PROGRAM SP3_2_Y131
VAR
	CompareOutput131_00: CMP_OC_DW;
	CompareOutput131_01: CMP_OC_DW;
	CompareOutput131_02: CMP_OC_DW;
	CompareOutput131_03: CMP_OC_DW;
	CompareOutput131_04: CMP_OC_DW;
	CompareOutput131_05: CMP_OC_DW;
	CompareOutput131_06: CMP_OC_DW;
	CompareOutput131_07: CMP_OC_DW;
	CompareOutput131_08: CMP_OC_DW;
	CompareOutput131_09: CMP_OC_DW;
	CompareOutput131_10: CMP_OC_DW;
	CompareOutput131_11: CMP_OC_DW;
	CompareOutput131_12: CMP_OC_DW;
	CompareOutput131_13: CMP_OC_DW;
	CompareOutput131_14: CMP_OC_DW;
	CompareOutput131_15: CMP_OC_DW;

END_VAR

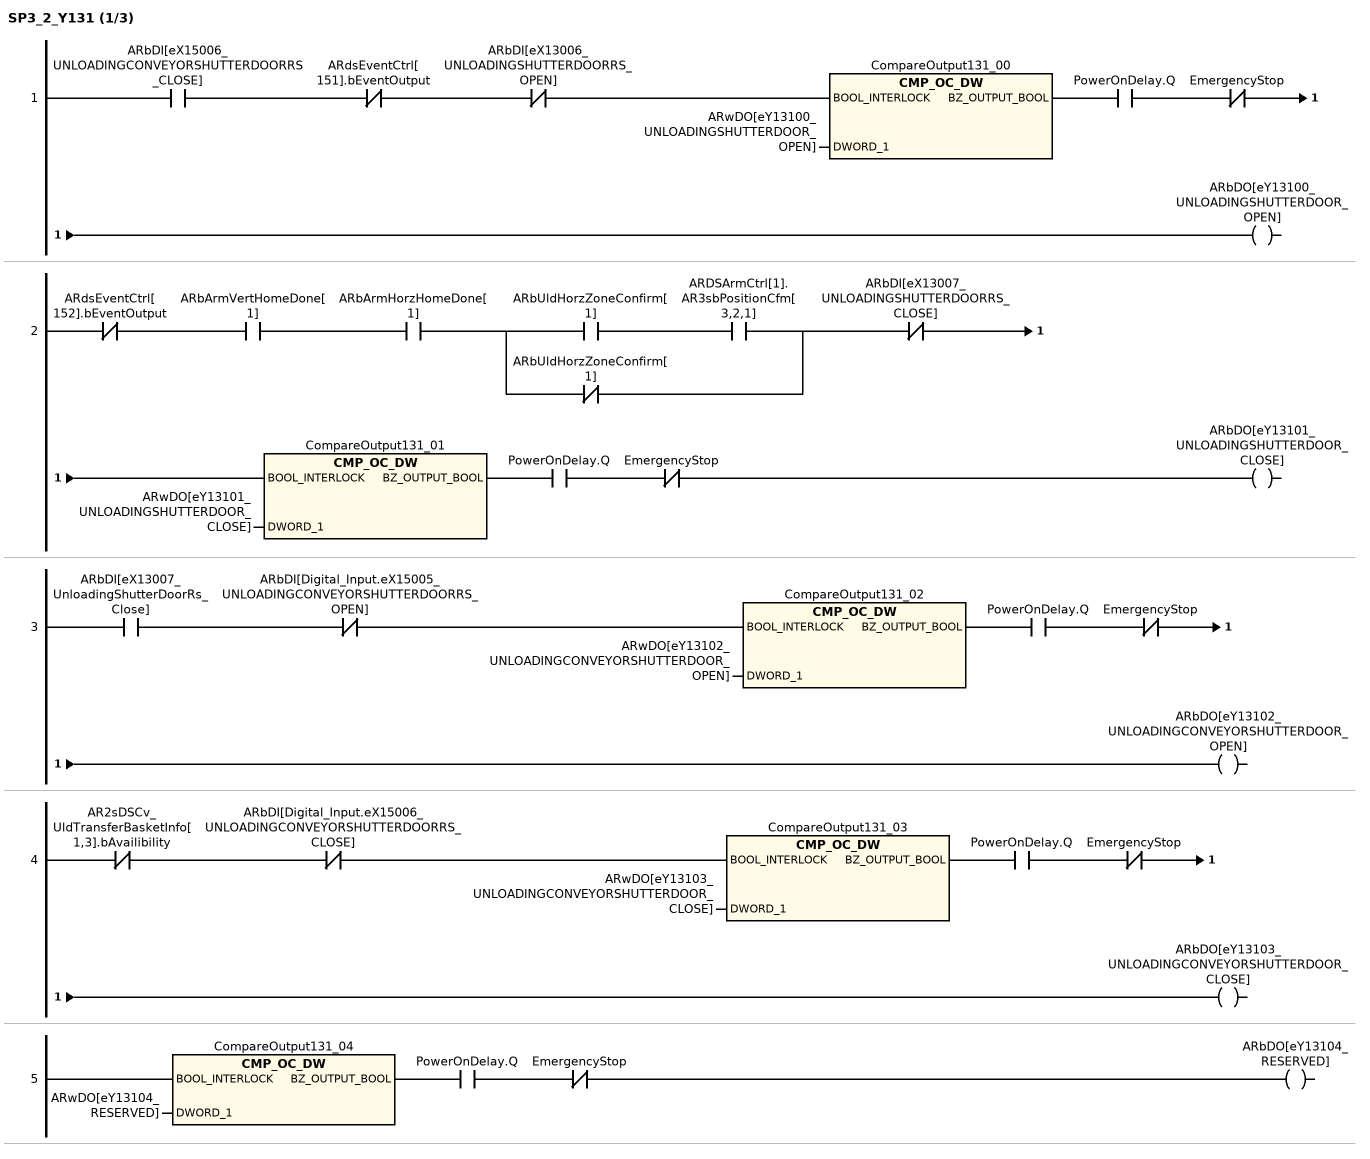
// NETWORK 1
CompareOutput131_00(BOOL_INTERLOCK := ARbDI[eX15006_UNLOADINGCONVEYORSHUTTERDOORRS_CLOSE] AND NOT ARdsEventCtrl[151].bEventOutput AND NOT ARbDI[eX13006_UNLOADINGSHUTTERDOORRS_OPEN], DWORD_1 := ARwDO[eY13100_UNLOADINGSHUTTERDOOR_OPEN]); // CMP_OC_DW
ARbDO[eY13100_UNLOADINGSHUTTERDOOR_OPEN] := CompareOutput131_00.BZ_OUTPUT_BOOL AND PowerOnDelay.Q AND NOT EmergencyStop;

// NETWORK 2
CompareOutput131_01(BOOL_INTERLOCK := NOT ARdsEventCtrl[152].bEventOutput AND ARbArmVertHomeDone[1] AND ARbArmHorzHomeDone[1] AND (ARbUldHorzZoneConfirm[1] AND ARDSArmCtrl[1].AR3sbPositionCfm[3,2,1] OR NOT ARbUldHorzZoneConfirm[1]) AND NOT ARbDI[eX13007_UNLOADINGSHUTTERDOORRS_CLOSE], DWORD_1 := ARwDO[eY13101_UNLOADINGSHUTTERDOOR_CLOSE]); // CMP_OC_DW
ARbDO[eY13101_UNLOADINGSHUTTERDOOR_CLOSE] := CompareOutput131_01.BZ_OUTPUT_BOOL AND PowerOnDelay.Q AND NOT EmergencyStop;

// NETWORK 3
CompareOutput131_02(BOOL_INTERLOCK := ARbDI[eX13007_UnloadingShutterDoorRs_Close] AND NOT ARbDI[Digital_Input.eX15005_UNLOADINGCONVEYORSHUTTERDOORRS_OPEN], DWORD_1 := ARwDO[eY13102_UNLOADINGCONVEYORSHUTTERDOOR_OPEN]); // CMP_OC_DW
ARbDO[eY13102_UNLOADINGCONVEYORSHUTTERDOOR_OPEN] := CompareOutput131_02.BZ_OUTPUT_BOOL AND PowerOnDelay.Q AND NOT EmergencyStop;

// NETWORK 4
CompareOutput131_03(BOOL_INTERLOCK := NOT AR2sDSCv_UldTransferBasketInfo[1,3].bAvailibility AND NOT ARbDI[Digital_Input.eX15006_UNLOADINGCONVEYORSHUTTERDOORRS_CLOSE], DWORD_1 := ARwDO[eY13103_UNLOADINGCONVEYORSHUTTERDOOR_CLOSE]); // CMP_OC_DW
ARbDO[eY13103_UNLOADINGCONVEYORSHUTTERDOOR_CLOSE] := CompareOutput131_03.BZ_OUTPUT_BOOL AND PowerOnDelay.Q AND NOT EmergencyStop;

// NETWORK 5
CompareOutput131_04(BOOL_INTERLOCK := TRUE, DWORD_1 := ARwDO[eY13104_RESERVED]); // CMP_OC_DW
ARbDO[eY13104_RESERVED] := CompareOutput131_04.BZ_OUTPUT_BOOL AND PowerOnDelay.Q AND NOT EmergencyStop;

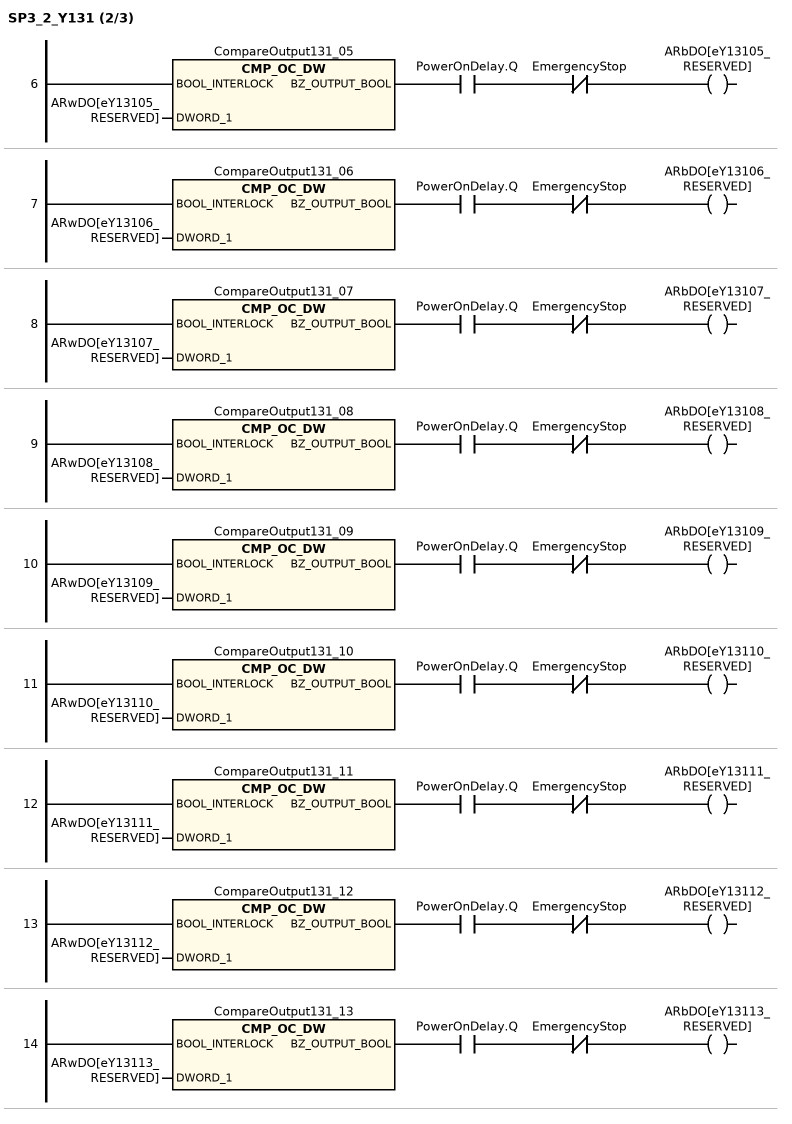
// NETWORK 6
CompareOutput131_05(BOOL_INTERLOCK := TRUE, DWORD_1 := ARwDO[eY13105_RESERVED]); // CMP_OC_DW
ARbDO[eY13105_RESERVED] := CompareOutput131_05.BZ_OUTPUT_BOOL AND PowerOnDelay.Q AND NOT EmergencyStop;

// NETWORK 7
CompareOutput131_06(BOOL_INTERLOCK := TRUE, DWORD_1 := ARwDO[eY13106_RESERVED]); // CMP_OC_DW
ARbDO[eY13106_RESERVED] := CompareOutput131_06.BZ_OUTPUT_BOOL AND PowerOnDelay.Q AND NOT EmergencyStop;

// NETWORK 8
CompareOutput131_07(BOOL_INTERLOCK := TRUE, DWORD_1 := ARwDO[eY13107_RESERVED]); // CMP_OC_DW
ARbDO[eY13107_RESERVED] := CompareOutput131_07.BZ_OUTPUT_BOOL AND PowerOnDelay.Q AND NOT EmergencyStop;

// NETWORK 9
CompareOutput131_08(BOOL_INTERLOCK := TRUE, DWORD_1 := ARwDO[eY13108_RESERVED]); // CMP_OC_DW
ARbDO[eY13108_RESERVED] := CompareOutput131_08.BZ_OUTPUT_BOOL AND PowerOnDelay.Q AND NOT EmergencyStop;

// NETWORK 10
CompareOutput131_09(BOOL_INTERLOCK := TRUE, DWORD_1 := ARwDO[eY13109_RESERVED]); // CMP_OC_DW
ARbDO[eY13109_RESERVED] := CompareOutput131_09.BZ_OUTPUT_BOOL AND PowerOnDelay.Q AND NOT EmergencyStop;

// NETWORK 11
CompareOutput131_10(BOOL_INTERLOCK := TRUE, DWORD_1 := ARwDO[eY13110_RESERVED]); // CMP_OC_DW
ARbDO[eY13110_RESERVED] := CompareOutput131_10.BZ_OUTPUT_BOOL AND PowerOnDelay.Q AND NOT EmergencyStop;

// NETWORK 12
CompareOutput131_11(BOOL_INTERLOCK := TRUE, DWORD_1 := ARwDO[eY13111_RESERVED]); // CMP_OC_DW
ARbDO[eY13111_RESERVED] := CompareOutput131_11.BZ_OUTPUT_BOOL AND PowerOnDelay.Q AND NOT EmergencyStop;

// NETWORK 13
CompareOutput131_12(BOOL_INTERLOCK := TRUE, DWORD_1 := ARwDO[eY13112_RESERVED]); // CMP_OC_DW
ARbDO[eY13112_RESERVED] := CompareOutput131_12.BZ_OUTPUT_BOOL AND PowerOnDelay.Q AND NOT EmergencyStop;

// NETWORK 14
CompareOutput131_13(BOOL_INTERLOCK := TRUE, DWORD_1 := ARwDO[eY13113_RESERVED]); // CMP_OC_DW
ARbDO[eY13113_RESERVED] := CompareOutput131_13.BZ_OUTPUT_BOOL AND PowerOnDelay.Q AND NOT EmergencyStop;

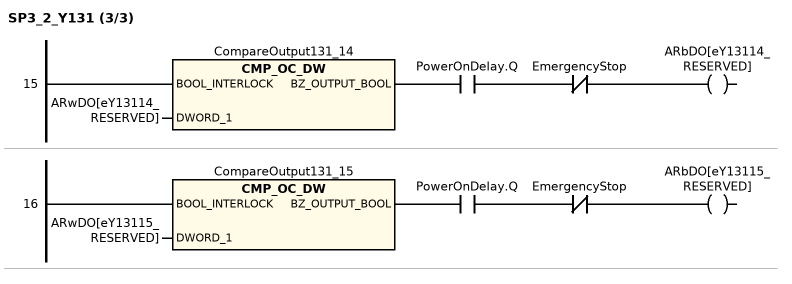
// NETWORK 15
CompareOutput131_14(BOOL_INTERLOCK := TRUE, DWORD_1 := ARwDO[eY13114_RESERVED]); // CMP_OC_DW
ARbDO[eY13114_RESERVED] := CompareOutput131_14.BZ_OUTPUT_BOOL AND PowerOnDelay.Q AND NOT EmergencyStop;

// NETWORK 16
CompareOutput131_15(BOOL_INTERLOCK := TRUE, DWORD_1 := ARwDO[eY13115_RESERVED]); // CMP_OC_DW
ARbDO[eY13115_RESERVED] := CompareOutput131_15.BZ_OUTPUT_BOOL AND PowerOnDelay.Q AND NOT EmergencyStop;

END_PROGRAM

(* stored: Version 1.1.0.1, ProductVersion 3.1.4024.11
   POU SP3_2_Y131: Id {57367501-9203-43dd-bffc-f6b9e23b4508}, SpecialFunc None *)
